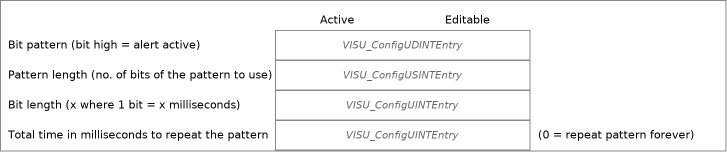
VISUALIZATION VISU_SafetyConfig_DomeAccessAlert  // 727x152
VAR_IN_OUT
    editable : SafetyDomeAccessAlertConfig;
	active : SafetyDomeAccessAlertConfig;
END_VAR
    Frame (275,30 255x30)
        shows VISU_ConfigUDINTEntry(active := active.pattern, editable := editable.pattern)
    Label (275,10 125x20), "Active"
    Label (405,10 125x20), "Editable"
    Label (5,30 285x30), "Bit pattern (bit high = alert active)"
    Frame (275,60 255x30)
        shows VISU_ConfigUSINTEntry(active := active.patternLength, editable := editable.patternLength)
    Label (5,60 285x30), "Pattern length (no. of bits of the pattern to use)"
    Frame (275,90 255x30)
        shows VISU_ConfigUINTEntry(active := active.bitLength, editable := editable.bitLength)
    Label (5,90 285x30), "Bit length (x where 1 bit = x milliseconds)"
    Frame (275,120 255x30)
        shows VISU_ConfigUINTEntry(active := active.totalTime, editable := editable.totalTime)
    Label (5,120 285x30), "Total time in milliseconds to repeat the pattern"
    Label (535,120 190x30), "(0 = repeat pattern forever)"
END_VISUALIZATION

(* stored: Version 1.1.0.1, ProductVersion 3.1.4019.2
   Visu VISU_SafetyConfig_DomeAccessAlert: Id {058d2599-0e73-4b01-8eb6-d48e1792975c} *)
